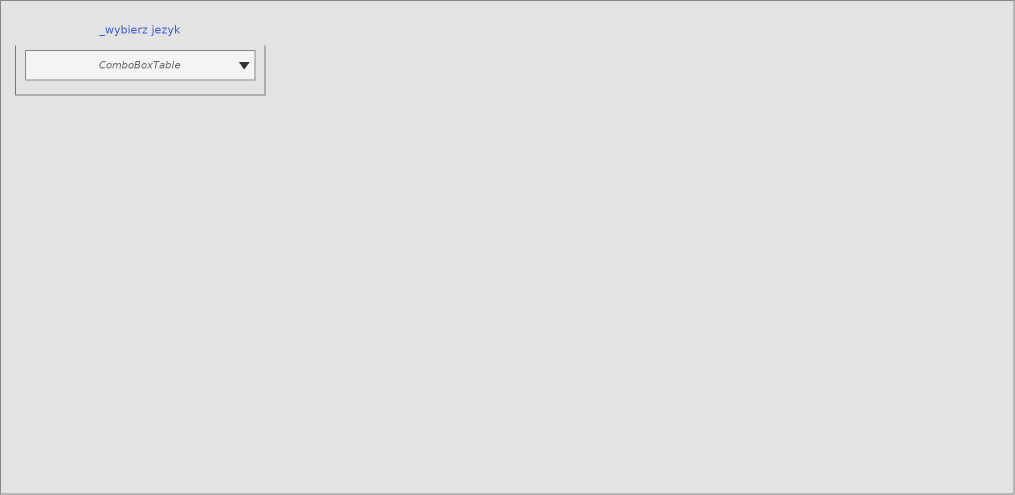
VISUALIZATION F_07_Settings  // 1015x495
VAR_IN_OUT
	stScreenData	: ST_MCHMIPrepareScreen_07_XX;

END_VAR
    Rectangle (15,15 250x80)
    Rectangle (15,15 250x30), "_wybierz jezyk", text list: 'TextList_07', text index: 0
    ComboBoxTable (25,50 230x30), variable: stScreenData.iChoosoLocation, data array: stScreenData.arrLocationDescription
        p3854506369: stScreenData.arrLocationDescription[INDEX]
        p1128707560: GVL_BaseConstans.NUMBER_OF_LOCATIONS -1
END_VISUALIZATION

(* stored: Version 1.1.0.1
   Visu F_07_Settings: Id {7806269d-d6e2-0719-05c5-824af7f14f54} *)
